      L     #t_Operator_Decision; // x1=Machine x/operator alarm
      L     1;
      ==I   ;
      S     #s_Decision_Data.Itm_Data.Process_1.EDS_Decision.Rejected_Operator;
      JC    MB10;

      L     #t_Operator_Decision; // x2=Machine x/operator clear
      L     2;
      ==I   ;
      S     #s_Decision_Data.Itm_Data.Process_1.EDS_Decision.Cleared_Operator;
      JC    MB10;

      L     #t_Operator_Decision; // x3=Machine x/operator unknown
      L     3;
      ==I   ;
      S     #s_Decision_Data.Itm_Data.Process_1.EDS_Decision.Operator_Unknown;
      JC    MB10;

      L     #t_Operator_Decision; // x4=Machine x/operator pending
      L     4;
      ==I   ;
      S     #s_Decision_Data.Itm_Data.Process_1.EDS_Decision.Operator_Pending;
      JC    MB10;

      L     #t_Operator_Decision; // x5=Machine x/operator timeout
      L     5;
      ==I   ;
      S     #s_Decision_Data.Itm_Data.Process_1.EDS_Decision.Timed_Out_Operator;
      JC    MB10;

      SET   ; // all other result are unknown
      S     #s_Decision_Data.Itm_Data.Process_1.EDS_Decision.Not_Analyzed;
      R     #s_Decision_Data.Itm_Data.Process_1.EDS_Decision.Cleared_Machine;
      R     #s_Decision_Data.Itm_Data.Process_1.EDS_Decision.Rejected_Machine;

MB10: AN    #s_Decision_Data.No_Decision_Expected;
      JCN   MB98;

      AN    #s_Decision_Data.Valid_LNK_Available;
      JCN   MB11; // Item already found, no data reload needed

      A(    ;
      L     #s_Decision_Data.Itm_Data.LNK;
      L     0;
      >I    ;
      )     ;
      JCN   MB12; // If LNK is unknown by EDS, start lookup on pseudo ID

      A(    ;
      L     #s_Decision_Data.Itm_Data.LNK;
      L     "DB_LNK_List".Entries_Present;
      <I    ;
      )     ;
      JCN   MB98; // If LNK is not in expected range: Abort data attachment

      CALL "FC_Read_ANY_Record" (// Read entire LNK record
           i_Record_Number          := #s_Decision_Data.Itm_Data.LNK,
           i_ANY_Data_Record        := "DB_UDT_LNK_Record",
           i_ANY_Data               := #s_Decision_Data.Itm_Data.LNK_Record,
           i_DB                     := "DB_LNK_List",
           i_DB_Event_Num           := #t_DB_Event_Num_Object);

      L     #s_Decision_Data.Itm_Data.LNK_Record.HBS;
      L     0;
      ==I   ;
      S     #s_Decision_Data.No_Decision_Expected;
      JC    MB98; // No HBS record = no screening result expected

MB11: CALL "FC_Read_Dint_Record" (
           i_Record_Number          := #s_Decision_Data.Itm_Data.LNK_Record.HBS,
           i_P_DINT_Record          := "DB_UDT_HBS_Record".HBS_Process_1.Screen_Result.Pseudo_ID,
           i_DB                     := "DB_HBS_List",
           i_DB_Event_Num           := #t_DB_Event_Num_Object,
           o_DINT                   := #t_HBS_Pseudo);

      L     #s_Decision_Data.Itm_Data.Pseudo;
      L     #t_HBS_Pseudo;
      ==D   ;
      JCN   MB12;

      CALL "FC_Read_ANY_Record" (
           i_Record_Number          := #s_Decision_Data.Itm_Data.LNK_Record.HBS,
           i_ANY_Data_Record        := "DB_UDT_HBS_Record".HBS_Process_1.ID_Screening,
           i_ANY_Data               := #s_HBS_Record_Screen_ID,
           i_DB                     := "DB_HBS_List",
           i_DB_Event_Num           := #t_DB_Event_Num_Object);

      L     #s_HBS_Record_Screen_ID;
      L     #i_HBO_ID;
      ==D   ;
      S     #s_Decision_Data.Valid_LNK_Available;
      R     #s_Decision_Data.Itm_Data.Process_1.No_Decision_Expected;
      JCN   MB12;

      JU    MB98;

MB12: A     #s_Decision_Data.Valid_LNK_Available;
      JC    MB98;

      SET   ;
      S     #s_Decision_Data.Inval_LNK_Pseudo_Lookup;

      L     L#0;
      L     #s_Decision_Data.Itm_Data.Pseudo;
      <>D   ;
      JCN   MB98; // If no pseudo available: End bag lookup, else: lookup bag by pseudo

      L     0;
      T     #t_Loop_Counter;

MB13: L     #t_Loop_Counter;
      JL    MB14;
      JU    MB20;
      JU    MB21;
      JU    MB22;
      JU    MB23;
      JU    MB24;
MB14: JU    MB98;
MB20: L     #s_EDS_Pseudo_Lookup.HBS_Lookup_Table[0];
      JU    MB30;
MB21: L     #s_EDS_Pseudo_Lookup.HBS_Lookup_Table[1];
      JU    MB30;
MB22: L     #s_EDS_Pseudo_Lookup.HBS_Lookup_Table[2];
      JU    MB30;
MB23: L     #s_EDS_Pseudo_Lookup.HBS_Lookup_Table[3];
      JU    MB30;
MB24: L     #s_EDS_Pseudo_Lookup.HBS_Lookup_Table[4];
      JU    MB30;
MB30: T     #t_HBS_Record_To_Check;
      L     0;
      >I    ;
      JCN   MB50;

      CALL "FC_Read_Dint_Record" (
           i_Record_Number          := #t_HBS_Record_To_Check,
           i_P_DINT_Record          := "DB_UDT_HBS_Record".HBS_Process_1.Screen_Result.Pseudo_ID,
           i_DB                     := "DB_HBS_List",
           i_DB_Event_Num           := #t_DB_Event_Num_Object,
           o_DINT                   := #t_HBS_Pseudo);

      L     #t_HBS_Pseudo;
      L     0;
      >D    ;
      JCN   MB39; // If HBS record still valid: continue check; If not: remove HBS from lookup table

      L     #t_HBS_Pseudo;
      L     #s_Decision_Data.Itm_Data.Pseudo;
      ==D   ;
      JCN   MB50; // If correct record is found: match record ID with machine, else: check next HBS record

      CALL "FC_Read_ANY_Record" (
           i_Record_Number          := #t_HBS_Record_To_Check,
           i_ANY_Data_Record        := "DB_UDT_HBS_Record".HBS_Process_1.ID_Screening,
           i_ANY_Data               := #s_HBS_Record_Screen_ID,
           i_DB                     := "DB_HBS_List",
           i_DB_Event_Num           := #t_DB_Event_Num_Object);

      L     #s_HBS_Record_Screen_ID;
      L     #i_HBO_ID;
      ==D   ;
      JCN   MB39; // If record was created at current machine: check LNK, else: check next HBS record

      CALL "FC_Read_Int_Record" (
           i_Record_Number          := #t_HBS_Record_To_Check,
           i_P_INT_Record           := "DB_UDT_HBS_Record".LNK,
           i_DB                     := "DB_HBS_List",
           i_DB_Event_Num           := #t_DB_Event_Num_Object,
           o_INT                    := #s_Decision_Data.Itm_Data.LNK);

      L     #s_Decision_Data.Itm_Data.LNK;
      L     0;
      <>I   ;
      JCN   MB39; // If a valid LNK is found by comparing pseudo ID's, process decision

      CALL "FC_Read_ANY_Record" (// Read entire LNK record
           i_Record_Number          := #s_Decision_Data.Itm_Data.LNK,
           i_ANY_Data_Record        := "DB_UDT_LNK_Record",
           i_ANY_Data               := #s_Decision_Data.Itm_Data.LNK_Record,
           i_DB                     := "DB_LNK_List",
           i_DB_Event_Num           := #t_DB_Event_Num_Object);

      L     #s_Decision_Data.Itm_Data.LNK_Record.HBS;
      L     #t_HBS_Record_To_Check;
      ==I   ;
      S     #s_Decision_Data.Valid_LNK_Available; // Valid LNK found through pseudo ID lookup
      R     #s_Decision_Data.Itm_Data.Process_1.No_Decision_Expected;

      JU    MB98;

MB39: L     #t_Loop_Counter;
      JL    MB40;
      JU    MB41;
      JU    MB42;
      JU    MB43;
      JU    MB44;
      JU    MB45;
MB40: JU    MB98;
MB41: L     0;
      T     #s_EDS_Pseudo_Lookup.HBS_Lookup_Table[0];
      JU    MB50;
MB42: L     0;
      T     #s_EDS_Pseudo_Lookup.HBS_Lookup_Table[1];
      JU    MB50;
MB43: L     0;
      T     #s_EDS_Pseudo_Lookup.HBS_Lookup_Table[2];
      JU    MB50;
MB44: L     0;
      T     #s_EDS_Pseudo_Lookup.HBS_Lookup_Table[3];
      JU    MB50;
MB45: L     0;
      T     #s_EDS_Pseudo_Lookup.HBS_Lookup_Table[4];
      JU    MB50;

MB50: AN    #s_Decision_Data.Valid_LNK_Available;
      JCN   MB98; // If correct LNK not found yet, try next pseudo

      L     #t_Loop_Counter;
      L     1;
      +I    ;
      T     #t_Loop_Counter;
      L     4;
      >I    ;
      JCN   MB13; // If not all records checked yet: loop; else: end lookup

MB98: A     #s_Decision_Data.Itm_Data.Process_1.No_Decision_Expected;
      O     #s_Decision_Data.No_Decision_Expected;
      AN    #s_Decision_Data.Itm_Data.Process_1.EDS_Decision.No_Decision;
      AN    #s_Decision_Data.Itm_Data.Process_1.EDS_Decision.Forced_Reject; // We already know the item is no longer present
      JCN   MB99; // Unable to find applicable item or item is not pending while decision is present: log event

      CALL "BLKMOV" (
           SRCBLK                   := #s_ISD_ID_Decision,// Log item data coming from EDS
           RET_VAL                  := #t_INT_not_used,
           DSTBLK                   := "DB_Outgoing_Msgs".Logging.MessageBody);

      CALL "FC_Snd_Log_Txt_Msg" (// 2602 Log_Message with the received data from the EDS
           i_ID                     := #i_HBO_ID,
           i_Event_value            := 2);// Unique identifier for decision proces

MB99: NOP   0;
NETWORK
TITLE =NA: Upd. PROCESS_1 records (HBS/LIC) upon decision + PackageRep
//Update local bag records to match received decisions
      A     #s_OS_New_Decision_Avail;
      O     #s_OS_Receive_Bag_Data;
      A     #s_Decision_Data.Valid_LNK_Available;
      JCN   NA99;

      AN    #s_Decision_Data.Itm_Data.Process_1.No_Decision_Expected;
      JCN   NA99; // If no HBS record available: stop receival, else: process

      L     #s_Decision_Data.Itm_Data.LNK_Record.LIC;
      L     0;
      <=I   ;
      S     #s_Decision_Data.LIC_Missing;

      CALL "FC_Read_ANY_Record" (
           i_Record_Number          := #s_Decision_Data.Itm_Data.LNK_Record.HBS,
           i_ANY_Data_Record        := "DB_UDT_HBS_Record",
           i_ANY_Data               := #s_Decision_Data.Itm_Data.HBS_Record,
           i_DB                     := "DB_HBS_List",
           i_DB_Event_Num           := #t_DB_Event_Num_Object);

      AN    #s_Decision_Data.Itm_Data.HBS_Record.HBS_Process_1.Result_Pending;
      ON    #s_Decision_Data.Itm_Data.HBS_Record.HBS_Process_1.Process_Active;
      O     #s_Decision_Data.Itm_Data.HBS_Record.HBS_General.Item_Lost;
      O(    ;
      L     #s_Decision_Data.Itm_Data.HBS_Record.HBS_Process_1.HBA_LNK;
      L     #s_Decision_Data.Itm_Data.LNK;
      <>I   ;
      )     ;
      S     #s_Decision_Data.Itm_Data.Process_1.No_Decision_Expected; // No decision expected concluded by HBS record content

      A     #s_Decision_Data.Itm_Data.Process_1.No_Decision_Expected;
      O     #s_Decision_Data.Itm_Data.Process_1.EDS_Decision.No_Decision;
      JC    NA22; // If process 1 decision expected and present: process, else: make sure PackageReport DB is empty

      A     #s_Decision_Data.Itm_Data.Process_1.EDS_Decision.Cleared_Machine;
      AN    #s_Decision_Data.Itm_Data.HBS_Record.HBS_Process_1.Machine_Result_Rcvd;
      JCN   NA01;

      L     1; // Update screening status : "CLEAR"
      T     #s_Decision_Data.Itm_Data.Process_1.Machine_Result_To_HL;

      L     1; // Clear
      T     #s_Decision_Data.Itm_Data.HBS_Record.HBS_Process_1.Bag_Status;

      SET   ;
      S     #s_Decision_Data.Itm_Data.HBS_Record.HBS_Process_1.Screen_Result.Reached_Screen_Level_1;

NA01: A     #s_Decision_Data.Itm_Data.Process_1.EDS_Decision.Rejected_Machine;
      AN    #s_Decision_Data.Itm_Data.HBS_Record.HBS_Process_1.Machine_Result_Rcvd;
      JCN   NA02;

      L     6; // Uncleared
      T     #s_Decision_Data.Itm_Data.Process_1.Machine_Result_To_HL;

      L     2; // Suspect
      T     #s_Decision_Data.Itm_Data.HBS_Record.HBS_Process_1.Bag_Status;

      SET   ;
      S     #s_Decision_Data.Itm_Data.HBS_Record.HBS_Process_1.Screen_Result.Failed_Screen_Level_1;

NA02: A     #s_Decision_Data.Itm_Data.Process_1.EDS_Decision.Not_Analyzed;
      JCN   NA04;

      L     #s_Decision_Data.Itm_Data.HBS_Record.HBS_Process_1.Bag_Status;
      L     4; // No Decision
      ==I   ;
      JCN   NA03;

      L     6;
      T     #s_Decision_Data.Itm_Data.Process_1.Machine_Result_To_HL;

      L     2; // Suspect
      T     #s_Decision_Data.Itm_Data.HBS_Record.HBS_Process_1.Bag_Status;

      SET   ;
      S     #s_Decision_Data.Itm_Data.HBS_Record.HBS_Process_1.Screen_Result.Failed_Screen_Level_1;

      JU    NA04;

NA03: L     6;
      T     #s_Decision_Data.Itm_Data.Process_1.Machine_Result_To_HL;

      L     4; // Not screened/Not Analyzed
      T     #s_Decision_Data.Itm_Data.HBS_Record.HBS_Process_1.Bag_Status;

NA04: A     #s_Decision_Data.Itm_Data.Process_1.EDS_Decision.Spacing_Error;
      JCN   NA06;

// Check current bag status for result
      L     #s_Decision_Data.Itm_Data.HBS_Record.HBS_Process_1.Bag_Status;
      L     4; // No Decision
      ==I   ;
      JCN   NA05;

      L     6;
      T     #s_Decision_Data.Itm_Data.Process_1.Machine_Result_To_HL;

      L     2; // Suspect
      T     #s_Decision_Data.Itm_Data.HBS_Record.HBS_Process_1.Bag_Status;

      SET   ;
      S     #s_Decision_Data.Itm_Data.HBS_Record.HBS_Process_1.Screen_Result.Failed_Screen_Level_1;

      JU    NA06;

NA05: L     6;
      T     #s_Decision_Data.Itm_Data.Process_1.Machine_Result_To_HL;

      L     4; // Not screened/Not Analyzed
      T     #s_Decision_Data.Itm_Data.HBS_Record.HBS_Process_1.Bag_Status;

NA06: A     #s_Decision_Data.Itm_Data.Process_1.EDS_Decision.Cleared_Operator; // Evaluate L2 (operator) decision
      AN    #s_Decision_Data.Itm_Data.HBS_Record.HBS_Process_1.Operator_Result_Rcvd;
      JCN   NA07; // L2 clear

      L     1; // Update screening status : "CLEAR"
      T     #s_Decision_Data.Itm_Data.Process_1.Operator_Result_To_HL;

      L     1; // Clear
      T     #s_Decision_Data.Itm_Data.HBS_Record.HBS_Process_1.Bag_Status;

      SET   ;
      S     #s_Decision_Data.Itm_Data.HBS_Record.HBS_Process_1.Screen_Result.Reached_Screen_Level_2;

NA07: A     #s_Decision_Data.Itm_Data.Process_1.EDS_Decision.Rejected_Operator; // L2 fail
      AN    #s_Decision_Data.Itm_Data.HBS_Record.HBS_Process_1.Operator_Result_Rcvd;
      JCN   NA08;

      L     6; // Update screening status : "REJECT"
      T     #s_Decision_Data.Itm_Data.Process_1.Operator_Result_To_HL;

      L     2; // Suspect
      T     #s_Decision_Data.Itm_Data.HBS_Record.HBS_Process_1.Bag_Status;

      SET   ;
      S     #s_Decision_Data.Itm_Data.HBS_Record.HBS_Process_1.Screen_Result.Failed_Screen_Level_2;

NA08: A     #s_Decision_Data.Itm_Data.Process_1.EDS_Decision.Timed_Out_Operator;
      AN    #s_Decision_Data.Itm_Data.HBS_Record.HBS_Process_1.Operator_Result_Rcvd;
      JCN   NA09;

      L     6;
      T     #s_Decision_Data.Itm_Data.Process_1.Operator_Result_To_HL;

      L     5; // OSR Time-Out
      T     #s_Decision_Data.Itm_Data.HBS_Record.HBS_Process_1.Bag_Status;

NA09: A     #s_Decision_Data.Itm_Data.Process_1.EDS_Decision.Operator_Pending;
      JCN   NA10;

      L     3; // Pending
      T     #s_Decision_Data.Itm_Data.HBS_Record.HBS_Process_1.Bag_Status;

NA10: A     #s_Decision_Data.Itm_Data.Process_1.EDS_Decision.Obvious_Threat;
      AN    #s_Decision_Data.Itm_Data.HBS_Record.HBS_Process_1.Operator_Result_Rcvd;
      JCN   NA11; // Obvious threat

      L     6;
      T     #s_Decision_Data.Itm_Data.Process_1.Operator_Result_To_HL;

      L     2; // Suspect
      T     #s_Decision_Data.Itm_Data.HBS_Record.HBS_Process_1.Bag_Status;

      SET   ;
      S     #s_Decision_Data.Itm_Data.HBS_Record.HBS_Process_1.Screen_Result.Failed_Screen_Level_2;

NA11: A     #s_Decision_Data.Itm_Data.Process_1.EDS_Decision.Forced_Reject;
      JCN   NA12; // No record updates, only log message

      CALL "FC_Write_Event" (// Log: Screening: Force reject on item
           i_Message_ID             := 3813,
           i_Event_value            := 0,
           i_DB_Event_Num           := #t_DB_Event_Num_Object,
           o_Return_Value           := #t_INT_not_used);

NA12: A     #s_Decision_Data.Itm_Data.Process_1.EDS_Decision.Operator_Unknown;
      AN    #s_Decision_Data.Itm_Data.HBS_Record.HBS_Process_1.Operator_Result_Rcvd;
      JCN   NA20;

      L     6;
      T     #s_Decision_Data.Itm_Data.Process_1.Operator_Result_To_HL;

NA20: A     #s_Decision_Data.Itm_Data.Process_1.EDS_Decision.Cleared_Machine;
      O     #s_Decision_Data.Itm_Data.Process_1.EDS_Decision.Rejected_Machine;
      O     #s_Decision_Data.Itm_Data.Process_1.EDS_Decision.Not_Analyzed;
      O     #s_Decision_Data.Itm_Data.Process_1.EDS_Decision.Spacing_Error;
      O     #s_Decision_Data.Itm_Data.Process_1.EDS_Decision.Cleared_Operator;
      O     #s_Decision_Data.Itm_Data.Process_1.EDS_Decision.Rejected_Operator;
      O     #s_Decision_Data.Itm_Data.Process_1.EDS_Decision.Timed_Out_Operator;
      O     #s_Decision_Data.Itm_Data.Process_1.EDS_Decision.Operator_Pending;
      O     #s_Decision_Data.Itm_Data.Process_1.EDS_Decision.Obvious_Threat;
      O     #s_Decision_Data.Itm_Data.Process_1.EDS_Decision.Operator_Unknown;
      JCN   NA99; // In case of new data: Update HBS, LIC and send PackageReport

      CALL "FC_Write_ANY_Record" (
           i_Record_Number          := #s_Decision_Data.Itm_Data.LNK_Record.HBS,
           i_ANY_Data_Record        := "DB_UDT_HBS_Record".HBS_Process_1.Screen_Result,
           i_ANY_Data               := #s_Decision_Data.Itm_Data.HBS_Record.HBS_Process_1.Screen_Result,
           i_DB                     := "DB_HBS_List",
           i_DB_Event_Num           := #t_DB_Event_Num_Object);

      CALL "FC_Write_Int_Record" (
           i_Record_Number          := #s_Decision_Data.Itm_Data.LNK_Record.HBS,
           i_P_INT_Record           := "DB_UDT_HBS_Record".HBS_Process_1.Bag_Status,
           i_DB                     := "DB_HBS_List",
           i_INT                    := #s_Decision_Data.Itm_Data.HBS_Record.HBS_Process_1.Bag_Status,
           i_DB_Event_Num           := #t_DB_Event_Num_Object);

      CALL "FC_Write_Event" (// Inform screening maintain functionality a HBS record update took place
           i_Message_ID             := 1,// Process number
           i_Event_value            := #s_Decision_Data.Itm_Data.LNK,
           i_DB_Event_Num           := #t_DB_Event_Pend_Num,
           o_Return_Value           := #t_INT_not_used);

      AN    #s_Decision_Data.LIC_Missing;
      JCN   NA22;

      CALL "FC_Write_ANY_Record" (
           i_Record_Number          := #s_Decision_Data.Itm_Data.LNK_Record.LIC,
           i_ANY_Data_Record        := "DB_UDT_LIC_Record".BIR.Process_1,
           i_ANY_Data               := #s_Decision_Data.Itm_Data.HBS_Record.HBS_Process_1.Screen_Result,
           i_DB                     := "DB_LIC_List",
           i_DB_Event_Num           := #t_DB_Event_Num_Object);

      CALL "FC_Write_Int_Record" (
           i_Record_Number          := #s_Decision_Data.Itm_Data.LNK_Record.LIC,
           i_P_INT_Record           := "DB_UDT_LIC_Record".BIR.Bag_Status,
           i_DB                     := "DB_LIC_List",
           i_INT                    := #s_Decision_Data.Itm_Data.HBS_Record.HBS_Process_1.Bag_Status,
           i_DB_Event_Num           := #t_DB_Event_Num_Object);

NA22: L     0;
      T     "DB_HBS_Results".Process_1.Level_1;
      T     "DB_HBS_Results".Process_1.Level_2;
      T     "DB_HBS_Results".Process_1.Level_3;
      T     "DB_HBS_Results".Process_1.Level_4;
      T     "DB_HBS_Results".Process_1.Level_5;

      L     #s_Decision_Data.Itm_Data.Process_1.Machine_Result_To_HL;
      L     0;
      >I    ;
      S     #s_Decision_Data.Send_Package_Report;
      JCN   NA23;

      L     #s_Decision_Data.Itm_Data.Process_1.Machine_Result_To_HL;
      T     "DB_HBS_Results".Process_1.Level_1; // Info for DAT layer

      CALL "FC_Write_BOOL_Record" (
           i_Record_Number          := #s_Decision_Data.Itm_Data.LNK_Record.HBS,
           i_P_BOOL_Record          := "DB_UDT_HBS_Record".HBS_Process_1.Machine_Result_Rcvd,
           i_DB                     := "DB_HBS_List",
           i_BOOL                   := TRUE,
           i_DB_Event_Num           := #t_DB_Event_Num_Object);

      A     #s_Decision_Data.Itm_Data.Process_1.EDS_Decision.Not_Analyzed;
      O     #s_Decision_Data.Itm_Data.Process_1.EDS_Decision.Cleared_Machine;
      O     #s_Decision_Data.Itm_Data.Process_1.EDS_Decision.Spacing_Error;
      O     #s_Decision_Data.Itm_Data.Process_1.EDS_Decision.Forced_Reject;
      JCN   NA23;

      CALL "FC_Write_BOOL_Record" (
           i_Record_Number          := #s_Decision_Data.Itm_Data.LNK_Record.HBS,
           i_P_BOOL_Record          := "DB_UDT_HBS_Record".HBS_Process_1.Result_Pending,
           i_DB                     := "DB_HBS_List",
           i_BOOL                   := FALSE,
           i_DB_Event_Num           := #t_DB_Event_Num_Object);

NA23: L     #s_Decision_Data.Itm_Data.Process_1.Operator_Result_To_HL;
      L     0;
      >I    ;
      S     #s_Decision_Data.Send_Package_Report;
      JCN   NA24;

      L     #s_Decision_Data.Itm_Data.Process_1.Operator_Result_To_HL;
      T     "DB_HBS_Results".Process_1.Level_2; // Info for DAT layer

      CALL "FC_Write_BOOL_Record" (
           i_Record_Number          := #s_Decision_Data.Itm_Data.LNK_Record.HBS,
           i_P_BOOL_Record          := "DB_UDT_HBS_Record".HBS_Process_1.Operator_Result_Rcvd,
           i_DB                     := "DB_HBS_List",
           i_BOOL                   := TRUE,
           i_DB_Event_Num           := #t_DB_Event_Num_Object);

      CALL "FC_Write_BOOL_Record" (
           i_Record_Number          := #s_Decision_Data.Itm_Data.LNK_Record.HBS,
           i_P_BOOL_Record          := "DB_UDT_HBS_Record".HBS_Process_1.Result_Pending,
           i_DB                     := "DB_HBS_List",
           i_BOOL                   := FALSE,
           i_DB_Event_Num           := #t_DB_Event_Num_Object);

NA24: A     #s_Decision_Data.Send_Package_Report;
      AN    #s_Decision_Data.Package_Report_Sent;
      JCN   NA99;

      CALL "FC_Write_Event" (
           i_Message_ID             := 1210,// Send PackageReport: Screening Result
           i_Event_value            := #s_Decision_Data.Itm_Data.LNK,
           i_DB_Event_Num           := #t_DB_Event_Num_Object,
           o_Return_Value           := #t_INT_not_used);

      SET   ;
      S     #s_Decision_Data.Package_Report_Sent;

NA99: NOP   0;

NETWORK
TITLE =OA: Update PROCESS_1 statisticals upon decision or timeout

      A     #s_OS_New_Decision_Avail;
      AN    #i_Test_Mode_Active; // Don't update machine decision statisticals in test mode
      JCN   OA99;

      A     #s_Decision_Data.Itm_Data.Process_1.EDS_Decision.Cleared_Machine;
      JCN   OA01;

      L     #s_Statisticals.R1.Count_Cleared;
      L     1;
      +I    ;
      T     #s_Statisticals.R1.Count_Cleared;

OA01: A     #s_Decision_Data.Itm_Data.Process_1.EDS_Decision.Rejected_Machine;
      JCN   OA02;

      L     #s_Statisticals.R1.Count_Rejected;
      L     1;
      +I    ;
      T     #s_Statisticals.R1.Count_Rejected;

OA02: A     #s_Decision_Data.Itm_Data.Process_1.EDS_Decision.Not_Analyzed;
      JCN   OA03;

      L     #s_Statisticals.R1.Count_NotAnalyzed;
      L     1;
      +I    ;
      T     #s_Statisticals.R1.Count_NotAnalyzed;

OA03: A     #s_Decision_Data.Itm_Data.Process_1.EDS_Decision.Cleared_Operator; // Evaluate L2 (operator) decision
      JCN   OA04; // L2 clear

      L     #s_Statisticals.R2.Count_Cleared;
      L     1;
      +I    ;
      T     #s_Statisticals.R2.Count_Cleared;

OA04: A     #s_Decision_Data.Itm_Data.Process_1.EDS_Decision.Rejected_Operator; // L2 fail
      JCN   OA05;

      L     #s_Statisticals.R2.Count_Rejected;
      L     1;
      +I    ;
      T     #s_Statisticals.R2.Count_Rejected;

OA05: A     #s_Decision_Data.Itm_Data.Process_1.EDS_Decision.Timed_Out_Operator;
      JCN   OA99;

      L     #s_Statisticals.R2.Count_TimeOut;
      L     1;
      +I    ;
      T     #s_Statisticals.R2.Count_TimeOut;

OA99: NOP   0;
NETWORK
TITLE =PA: Force reject
//When a bag decision is pending while it's no longer required. The bag will be
//force rejected
      CALL #s_FB_HBS_Force_Reject (
           i_ID                     := #i_HBO_ID,
           i_DB_Event               := #i_DB_Event_Object,
           i_DB_Fifo_Force_Reject   := #i_DB_Fifo_Force_Reject,
           i_Forced_Reject_Ack      := #i_IO_Forced_Reject_Ack,
           o_Force_Reject           := #o_IO_Force_Reject,
           o_Pseudo_Code_ForceRej   := #o_IO_Pseud_Code_ForceRej);

      A     #o_IO_Force_Reject;
      FP    #s_FP_Force_Reject;
      JCN   PA99;

      L     #s_Statisticals.Force_Rejected;
      L     1;
      +I    ;
      T     #s_Statisticals.Force_Rejected;

PA99: NOP   0;
NETWORK
TITLE =QA: Send and clear statisticals

      A     #i_CMD_Send_Stat;
      JCN   QA99;

      CALL "FC_Write_Event" (
           i_Message_ID             := 2001,
           i_Event_value            := #s_Statisticals.Bags_Handed_Over,
           i_DB_Event_Num           := #t_DB_Event_Num_Object,
           o_Return_Value           := #t_INT_not_used);

      CALL "FC_Write_Event" (
           i_Message_ID             := 2002,
           i_Event_value            := #s_Statisticals.Tracking.Positively_Tracked,
           i_DB_Event_Num           := #t_DB_Event_Num_Object,
           o_Return_Value           := #t_INT_not_used);

      CALL "FC_Write_Event" (
           i_Message_ID             := 2003,
           i_Event_value            := #s_Statisticals.Tracking.Trk_Lost_Result_Pending,
           i_DB_Event_Num           := #t_DB_Event_Num_Object,
           o_Return_Value           := #t_INT_not_used);

      CALL "FC_Write_Event" (
           i_Message_ID             := 2004,
           i_Event_value            := #s_Statisticals.Tracking.Trk_Lost_No_Result,
           i_DB_Event_Num           := #t_DB_Event_Num_Object,
           o_Return_Value           := #t_INT_not_used);

      CALL "FC_Write_Event" (
           i_Message_ID             := 2005,
           i_Event_value            := #s_Statisticals.R1.No_Decision_Required,
           i_DB_Event_Num           := #t_DB_Event_Num_Object,
           o_Return_Value           := #t_INT_not_used);

      CALL "FC_Write_Event" (
           i_Message_ID             := 2006,
           i_Event_value            := #s_Statisticals.R1.Count_Cleared,
           i_DB_Event_Num           := #t_DB_Event_Num_Object,
           o_Return_Value           := #t_INT_not_used);

      CALL "FC_Write_Event" (
           i_Message_ID             := 2007,
           i_Event_value            := #s_Statisticals.R1.Count_Rejected,
           i_DB_Event_Num           := #t_DB_Event_Num_Object,
           o_Return_Value           := #t_INT_not_used);

      CALL "FC_Write_Event" (
           i_Message_ID             := 2008,
           i_Event_value            := #s_Statisticals.R2.Count_Cleared,
           i_DB_Event_Num           := #t_DB_Event_Num_Object,
           o_Return_Value           := #t_INT_not_used);

      CALL "FC_Write_Event" (
           i_Message_ID             := 2009,
           i_Event_value            := #s_Statisticals.R2.Count_Rejected,
           i_DB_Event_Num           := #t_DB_Event_Num_Object,
           o_Return_Value           := #t_INT_not_used);

      CALL "FC_Write_Event" (
           i_Message_ID             := 2010,
           i_Event_value            := #s_Statisticals.R2.Count_TimeOut,
           i_DB_Event_Num           := #t_DB_Event_Num_Object,
           o_Return_Value           := #t_INT_not_used);

      CALL "FC_Write_Event" (
           i_Message_ID             := 2011,
           i_Event_value            := #s_Statisticals.R1.Count_NotAnalyzed,
           i_DB_Event_Num           := #t_DB_Event_Num_Object,
           o_Return_Value           := #t_INT_not_used);

      CALL "FC_Write_Event" (
           i_Message_ID             := 2012,
           i_Event_value            := #s_Statisticals.Force_Rejected,
           i_DB_Event_Num           := #t_DB_Event_Num_Object,
           o_Return_Value           := #t_INT_not_used);

      L     0;
      T     #s_Statisticals.Bags_Handed_Over;
      T     #s_Statisticals.R1.Count_Cleared;
      T     #s_Statisticals.R2.Count_Cleared;
      T     #s_Statisticals.R1.Count_Rejected;
      T     #s_Statisticals.R2.Count_Rejected;
      T     #s_Statisticals.R1.Count_NotAnalyzed;
      T     #s_Statisticals.R2.Count_TimeOut;
      T     #s_Statisticals.Tracking.Positively_Tracked;
      T     #s_Statisticals.Tracking.Trk_Lost_Result_Pending;
      T     #s_Statisticals.Tracking.Trk_Lost_No_Result;
      T     #s_Statisticals.Force_Rejected;
      T     #s_Statisticals.R1.No_Decision_Required;

QA99: NOP   0;
NETWORK
TITLE =RA: Date/Time Master Clock Designator

      CLR   ; // MV3D is master clock
      =     #o_IO_MasterClkDesignator; // No need to send BHS clock

      L     #i_IO_Time_Sync_Sec; // Seconds [00..59]
      T     #o_IO_Time_Sync_Sec;

      L     #i_IO_Time_Sync_Min; // Minutes [00..59]
      T     #o_IO_Time_Sync_Min;

      L     #i_IO_Time_Sync_Hour; // Time_hours [01..24]
      T     #o_IO_Time_Sync_Hour;

      L     #i_IO_Time_Sync_Day; // Day of month [1..31]
      T     #o_IO_Time_Sync_Day;

      L     #i_IO_Time_Sync_Month; // Month [1..31]
      T     #o_IO_Time_Sync_Month;

      L     #i_IO_Time_Sync_Year; // Year  [0..99]
      T     #o_IO_Time_Sync_Year;

NETWORK
TITLE =SA: Object/Section states
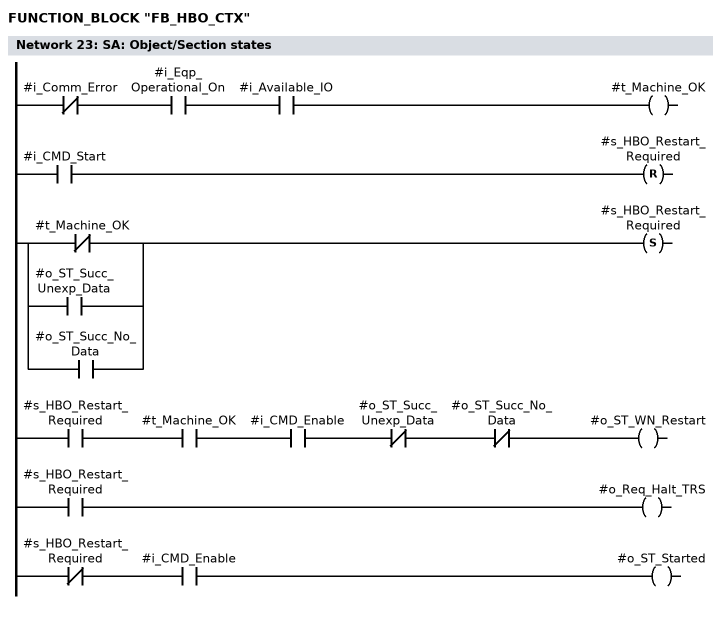

      AN    #i_Comm_Error;
      A     #i_Eqp_Operational_On;
      A     #i_Available_IO;
      =     #t_Machine_OK;

      A     #i_CMD_Start;
      R     #s_HBO_Restart_Required;

      AN    #t_Machine_OK;
      O     #o_ST_Succ_Unexp_Data;
      O     #o_ST_Succ_No_Data;
      S     #s_HBO_Restart_Required;

      A     #s_HBO_Restart_Required;
      A     #t_Machine_OK;
      A     #i_CMD_Enable;
      AN    #o_ST_Succ_Unexp_Data;
      AN    #o_ST_Succ_No_Data;
      =     #o_ST_WN_Restart;

      A     #s_HBO_Restart_Required;
      =     #o_Req_Halt_TRS;

      AN    #s_HBO_Restart_Required;
      A     #i_CMD_Enable;
      =     #o_ST_Started;
NETWORK
TITLE =TA: Copy BHS_ID.BAGIDARRAY (Data + IATA + PSEUDO) to output
//BHS_ID = BagIDArray + IATA + PSEUDO
      TAR2  #t_AR2_Store_Restore; // AR2 Store

      L     P##i_IO_BHS_ID; // 'area-crossing pointer'
      L     #t_Base_Address; // 'relative address'-mask
      +D    ;
      LAR1  ; // 'absolute address' Source
      LAR2  P##t_IO_BHS_ID; //  address Destination

      L     W [AR1,P#0.0]; // Copy ANY pointer
      T     LW [AR2,P#0.0]; // Byte0=$10 (for S7), Byte1=data type
      L     W [AR1,P#2.0];
      T     LW [AR2,P#2.0]; // Byte2..3=Repetition factor
      L     W [AR1,P#4.0];
      T     LW [AR2,P#4.0]; // Byte4..5=DB number
      L     D [AR1,P#6.0];
      T     LD [AR2,P#6.0]; // Byte6=memory area, Byte7..9=Byte,Bit address

      LAR2  #t_AR2_Store_Restore; // AR2 Restore

      CALL "BLKMOV" (
           SRCBLK                   := #s_BHS_ID,
           RET_VAL                  := #t_INT_not_used,
           DSTBLK                   := #t_IO_BHS_ID);

END_FUNCTION_BLOCK

